FUNCTION LogMessage : BOOL
VAR_INPUT
	msg : STRING;
	cleaning :BOOL;
END_VAR
VAR
END_VAR

IF GVL.Message <> msg THEN
GVL.Message := msg;
END_IF;
GVL.CLEANING := cleaning;
LogMessage := TRUE;

END_FUNCTION

(* stored: Version 1.1.0.1, ProductVersion 3.1.4024.15
   POU LogMessage: Id {800e1b71-e7e6-4a9c-9169-bf36698146e3}, SpecialFunc None *)
